PROGRAM TestRunner
VAR
	fbTestOTelMetricCore : FB_Test_OTelMetricCore;
END_VAR

TcUnit.Run();
fbTestOTelMetricCore();

END_PROGRAM

(* stored: Version 1.1.0.1
   POU TestRunner: Id {31f4ab78-3c98-459b-a21c-1adba1822291}, SpecialFunc None *)
